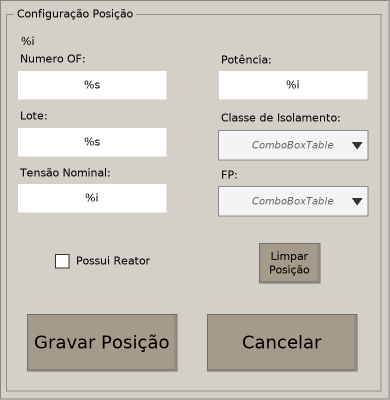
VISUALIZATION ConfigPosicao_3  // 390x400
VAR_IN_OUT
	bReator: BOOL;
	iOFnumber: INT;
	iSrlNumber: INT;
	
	
	
END_VAR
    GroupBox (6,6 375x385), "Configuração Posição"
        Checkbox (47,242 110x26), "Possui Reator", variable: gravarConfigPosicao021.bReator[2]
        Label (11,38 81x30), "Numero OF:"
        Textfield (11,64 150x30), "%s", text variable: GVL.cfgPos_OF021
            OnMouseDown: write the text variable via VisuDialogs.Numpad
        Label (11,152 103x30), "Tensão Nominal:"
        Button (21,308 150x57), "Gravar Posição"
            OnMouseClick: CloseDialog Dialog=ConfigPosicao_3, Result=OK, NumpadKeypadSet=True
            OnMouseClick: execute { gravarConfigPosicao021(); }
        Button (201,308 150x57), "Cancelar"
            OnMouseClick: CloseDialog Dialog=ConfigPosicao_3, Result=Cancel, NumpadKeypadSet=True
        Button (253,237 61x40), "Limpar Posição"
            OnMouseClick: CloseDialog Dialog=ConfigPosicao_3, Result=Cancel, NumpadKeypadSet=True
            OnMouseClick: execute {
                IF gvl_p.aPositionsE021[gvl.actPos].cor = 1
                OR gvl_p.aPositionsE021[gvl.actPos].cor = 2 THEN
                IF gvl.totalPos[2] > 0 THEN
                gvl.totalPos[2]:= gvl.totalPos[2]-1;
                END_IF
                END_IF
                gvl_p.aPositionsE021[gvl.actPos].numOF:='0';
                gvl_p.aPositionsE021[gvl.actPos].lote:='0';
                gvl_p.aPositionsE021[gvl.actPos].class:=0;
                gvl_p.aPositionsE021[gvl.actPos].pot:=0;
                gvl_p.aPositionsE021[gvl.actPos].cor:=0;
                gvl_p.aPositionsE021[gvl.actPos].text:='';
                bReator:=false;
                ///// GERADOR DE LOG -------------------------------------------------------------
                gvl.envialog:= 'Posição Nº ';
                gvl.envialog:= concat(gvl.envialog, INT_TO_STRING(gvl.actPos));
                gvl.envialog:= concat(gvl.envialog,' foi limpa. ESTUFA 021');
                gvl.logRegister21:= gvl.envialog;
            }
        Textfield (212,64 150x30), "%i", text variable: GVL.cfgPos_Pot021
            OnMouseDown: write the text variable via VisuDialogs.Numpad
        Label (11,95 81x30), "Lote:"
        Label (212,154 56x30), "FP:"
        Label (212,97 144x30), "Classe de Isolamento:"
        Textfield (11,177 150x30), "%i", text variable: GVL.cfgPos_Class021
            OnMouseDown: write the text variable via VisuDialogs.Numpad
    Label (218,45 56x30), "Potência:"
    Rectangle (17,30 22x23), "%i", text variable: GVL.actPos
    Textfield (17,127 150x30), "%s", text variable: GVL.cfgPos_LT021
        OnMouseDown: write the text variable via VisuDialogs.Keypad
    ComboBoxTable (218,130 150x30), variable: GVL.cfgPos_Iso021, data array: GVL_P.arr_Iso_3
        p3854506369: GVL_P.arr_Iso_3[INDEX]
    ComboBoxTable (218,186 150x30), variable: GVL.cfgPos_FP021, data array: GVL_P.arr_FP_3
        p3854506369: GVL_P.arr_FP_3[INDEX]
END_VISUALIZATION

(* stored: Version 1.1.0.1, ProductVersion 3.1.4024.12
   Visu ConfigPosicao_3: Id {4db39272-76fd-4a7f-8493-da50291a50d7} *)
